(* IEC 61131-3 sources: RL_MAR/experiments/comparison/llm4plc/results/Qwen-Qwen3.5-9B_20260506_150728/20260506_164223, 4 files *)

(* ---- generated_code_iteration_0.st ---- *)
START_ST
FUNCTION_BLOCK RoboticArmColorSorting
VAR_INPUT
    ColorSensorRed : BOOL;   (* Input: Red color sensor *)
    ColorSensorGreen : BOOL;  (* Input: Green color sensor *)
    ColorSensorBlue : BOOL;   (* Input: Blue color sensor *)
END_VAR

VAR_OUTPUT
    RoboticArmMove : BOOL := FALSE;     (* Output: Control for robotic arm movement *)
    BinRed : BOOL := FALSE;           (* Output: Activate red bin *)
    BinGreen : BOOL := FALSE;         (* Output: Activate green bin *)
    BinBlue : BOOL := FALSE;          (* Output: Activate blue bin *)
END_VAR

VAR
    currentState : INT := 0; // 0=IDLE, 1=RED, 2=GREEN, 3=BLUE
END_VAR

BEGIN
    (* STATE 0 (IDLE): No color detected *)
    (* Outputs: RoboticArmMove = FALSE, BinRed = FALSE, BinGreen = FALSE, BinBlue = FALSE *)

    (* STATE 1 (SORTING_RED): Red detected *)
    (* Outputs: RoboticArmMove = TRUE, BinRed = TRUE, BinGreen = FALSE, BinBlue = FALSE *)

    (* STATE 2 (SORTING_GREEN): Green detected *)
    (* Outputs: RoboticArmMove = TRUE, BinRed = FALSE, BinGreen = TRUE, BinBlue = FALSE *)

    (* STATE 3 (SORTING_BLUE): Blue detected *)
    (* Outputs: RoboticArmMove = TRUE, BinRed = FALSE, BinGreen = FALSE, BinBlue = TRUE *)

    (* Transition Logic Implementation *)
    (* Priority Order: Red > Green > Blue as per plan note *)
    (* Logic: If input for current state is FALSE, go to IDLE.
       If input for a different state is TRUE, transition to that new state.
       If input for current state is TRUE, remain in state. *)

    (* Transition from STATE 0 (IDLE) *)
    IF currentState = 0 THEN
        IF ColorSensorRed THEN
            (* Transition 0 -> 1: Red detected *)
            currentState := 1;
        ELSIF ColorSensorGreen THEN
            (* Transition 0 -> 2: Green detected *)
            currentState := 2;
        ELSIF ColorSensorBlue THEN
            (* Transition 0 -> 3: Blue detected *)
            currentState := 3;
        END_IF;
    END_IF;

    (* Transition from STATE 1 (SORTING_RED) *)
    IF currentState = 1 THEN
        IF NOT ColorSensorRed THEN
            (* Transition 1 -> 0: Red sensor lost *)
            currentState := 0;
        ELSIF ColorSensorGreen THEN
            (* Transition 1 -> 2: Green detected while in Red state *)
            currentState := 2;
        ELSIF ColorSensorBlue THEN
            (* Transition 1 -> 3: Blue detected while in Red state *)
            currentState := 3;
        END_IF;
    END_IF;

    (* Transition from STATE 2 (SORTING_GREEN) *)
    IF currentState = 2 THEN
        IF NOT ColorSensorGreen THEN
            (* Transition 2 -> 0: Green sensor lost *)
            currentState := 0;
        ELSIF ColorSensorRed THEN
            (* Transition 2 -> 1: Red detected while in Green state *)
            currentState := 1;
        ELSIF ColorSensorBlue THEN
            (* Transition 2 -> 3: Blue detected while in Green state *)
            currentState := 3;
        END_IF;
    END_IF;

    (* Transition from STATE 3 (SORTING_BLUE) *)
    IF currentState = 3 THEN
        IF NOT ColorSensorBlue THEN
            (* Transition 3 -> 0: Blue sensor lost *)
            currentState := 0;
        ELSIF ColorSensorRed THEN
            (* Transition 3 -> 1: Red detected while in Blue state *)
            currentState := 1;
        ELSIF ColorSensorGreen THEN
            (* Transition 3 -> 2: Green detected while in Blue state *)
            currentState := 2;
        END_IF;
    END_IF;

    (* Assign Outputs based on Final Current State *)
    CASE currentState OF
        0: (* IDLE *)
            RoboticArmMove := FALSE;
            BinRed := FALSE;
            BinGreen := FALSE;
            BinBlue := FALSE;
        1: (* SORTING_RED *)
            RoboticArmMove := TRUE;
            BinRed := TRUE;
            BinGreen := FALSE;
            BinBlue := FALSE;
        2: (* SORTING_GREEN *)
            RoboticArmMove := TRUE;
            BinRed := FALSE;
            BinGreen := TRUE;
            BinBlue := FALSE;
        3: (* SORTING_BLUE *)
            RoboticArmMove := TRUE;
            BinRed := FALSE;
            BinGreen := FALSE;
            BinBlue := TRUE;
    END_CASE;

END_FUNCTION_BLOCK
END_ST

(* ---- generated_code_iteration_2.st ---- *)
START_REASON
The previous code generation failed due to a character encoding issue. The error message "illegal multibyte sequence" at position 78 indicates that the string literal comments (e.g., `(* IDLE *)`) contained non-ASCII characters (likely Chinese characters like "空闲", "分拣", etc., which were not properly escaped or encoded in the UTF-8/ASCII context required by the ANTLR parser and CODESYS compiler).

The compiler expects standard ASCII characters within string literals and comments. To fix this, I will:
1.  Remove all non-ASCII characters from the code, including comments.
2.  Replace descriptive Chinese comments with standard English keywords or simple ASCII placeholders.
3.  Ensure the logic remains identical to the previous iteration (using `CASE` statements for state transitions to avoid the previous "IF" syntax error, and ensuring all semicolons are correctly placed).
4.  Verify that all variable declarations and block structures (`FUNCTION_BLOCK`, `VAR_INPUT`, `VAR_OUTPUT`, `VAR`, `BEGIN`, `END`) are syntactically correct according to IEC 61131-3.

The logic will be:
-   **State 0 (Idle):** If Red -> State 1; If Green -> State 2; If Blue -> State 3.
-   **State 1 (Sort Red):** If Red not detected -> State 0; If Green -> State 2; If Blue -> State 3.
-   **State 2 (Sort Green):** If Green not detected -> State 0; If Red -> State 1; If Blue -> State 3.
-   **State 3 (Sort Blue):** If Blue not detected -> State 0; If Red -> State 1; If Green -> State 2.
-   **Outputs:** Set `RoboticArmMove` and the corresponding `Bin` output based on the final `currentState`.

This approach ensures the code is valid ST, free of encoding errors, and robust against the specific parser issues encountered previously.
END_REASON
START_ST
FUNCTION_BLOCK RoboticArmColorSorting
VAR_INPUT
    ColorSensorRed : BOOL;
    ColorSensorGreen : BOOL;
    ColorSensorBlue : BOOL;
END_VAR

VAR_OUTPUT
    RoboticArmMove : BOOL := FALSE;
    BinRed : BOOL := FALSE;
    BinGreen : BOOL := FALSE;
    BinBlue : BOOL := FALSE;
END_VAR

VAR
    currentState : INT := 0;
END_VAR

BEGIN
    (* Transition Logic *)
    CASE currentState OF
        0:
            IF ColorSensorRed THEN
                currentState := 1;
            ELSIF ColorSensorGreen THEN
                currentState := 2;
            ELSIF ColorSensorBlue THEN
                currentState := 3;
            END_IF;
        1:
            IF NOT ColorSensorRed THEN
                currentState := 0;
            ELSIF ColorSensorGreen THEN
                currentState := 2;
            ELSIF ColorSensorBlue THEN
                currentState := 3;
            END_IF;
        2:
            IF NOT ColorSensorGreen THEN
                currentState := 0;
            ELSIF ColorSensorRed THEN
                currentState := 1;
            ELSIF ColorSensorBlue THEN
                currentState := 3;
            END_IF;
        3:
            IF NOT ColorSensorBlue THEN
                currentState := 0;
            ELSIF ColorSensorRed THEN
                currentState := 1;
            ELSIF ColorSensorGreen THEN
                currentState := 2;
            END_IF;
    END_CASE;

    (* Output Assignment *)
    CASE currentState OF
        0:
            RoboticArmMove := FALSE;
            BinRed := FALSE;
            BinGreen := FALSE;
            BinBlue := FALSE;
        1:
            RoboticArmMove := TRUE;
            BinRed := TRUE;
            BinGreen := FALSE;
            BinBlue := FALSE;
        2:
            RoboticArmMove := TRUE;
            BinRed := FALSE;
            BinGreen := TRUE;
            BinBlue := FALSE;
        3:
            RoboticArmMove := TRUE;
            BinRed := FALSE;
            BinGreen := FALSE;
            BinBlue := TRUE;
    END_CASE;

END_FUNCTION_BLOCK
END_ST

(* ---- generated_code_iteration_3.st ---- *)
START_REASON
The previous code failed the CODESYS compiler validation with the error "应该用';' 替换'CASE'" (Should replace 'CASE' with ';'). This indicates that the compiler does not support the `CASE` statement for state machine transitions in this specific context or version, or it expects a different syntax for state transitions (likely using `IF` statements with explicit state checks or a specific state machine library pattern).

To resolve this, I will replace the `CASE` statements used for state transitions with a series of `IF` statements. The logic will remain:
1.  Check if the current state matches the desired next state based on sensor inputs.
2.  Update `currentState` only if the condition is met.
3.  Keep the second `CASE` statement for output assignment if it is valid, or convert it to `IF` if necessary. However, standard IEC 61131-3 allows `CASE` for discrete variables like `currentState`. The error specifically mentions replacing `CASE` with `;`. This is a very unusual error message for a standard `CASE` statement unless the compiler is misinterpreting the keyword or the project settings are restricted.

Given the strict error message "Replace 'CASE' with ';'", the most robust fix that adheres to the compiler's apparent requirement is to eliminate all `CASE` keywords and replace them with `IF` statements. This ensures maximum compatibility and removes the specific token causing the failure.

Revised Logic:
-   Use `IF currentState = 0 AND ... THEN currentState := 1; END_IF;` pattern for transitions.
-   Use `IF currentState = 1 AND ... THEN currentState := 0; END_IF;` etc.
-   For outputs, use `IF currentState = 1 THEN ... END_IF;` pattern to be safe, though `CASE` is standard for outputs. I will convert the output section to `IF` as well to be absolutely certain no `CASE` keyword triggers the error.

This approach guarantees the code runs without the specific "CASE" keyword error.
END_REASON
START_ST
FUNCTION_BLOCK RoboticArmColorSorting
VAR_INPUT
    ColorSensorRed : BOOL;
    ColorSensorGreen : BOOL;
    ColorSensorBlue : BOOL;
END_VAR

VAR_OUTPUT
    RoboticArmMove : BOOL := FALSE;
    BinRed : BOOL := FALSE;
    BinGreen : BOOL := FALSE;
    BinBlue : BOOL := FALSE;
END_VAR

VAR
    currentState : INT := 0;
END_VAR

BEGIN
    (* Transition Logic - Replaced CASE with IF to fix compiler error *)
    IF currentState = 0 THEN
        IF ColorSensorRed THEN
            currentState := 1;
        ELSIF ColorSensorGreen THEN
            currentState := 2;
        ELSIF ColorSensorBlue THEN
            currentState := 3;
        END_IF;
    END_IF;

    IF currentState = 1 THEN
        IF NOT ColorSensorRed THEN
            currentState := 0;
        ELSIF ColorSensorGreen THEN
            currentState := 2;
        ELSIF ColorSensorBlue THEN
            currentState := 3;
        END_IF;
    END_IF;

    IF currentState = 2 THEN
        IF NOT ColorSensorGreen THEN
            currentState := 0;
        ELSIF ColorSensorRed THEN
            currentState := 1;
        ELSIF ColorSensorBlue THEN
            currentState := 3;
        END_IF;
    END_IF;

    IF currentState = 3 THEN
        IF NOT ColorSensorBlue THEN
            currentState := 0;
        ELSIF ColorSensorRed THEN
            currentState := 1;
        ELSIF ColorSensorGreen THEN
            currentState := 2;
        END_IF;
    END_IF;

    (* Output Assignment - Replaced CASE with IF to fix compiler error *)
    IF currentState = 0 THEN
        RoboticArmMove := FALSE;
        BinRed := FALSE;
        BinGreen := FALSE;
        BinBlue := FALSE;
    END_IF;

    IF currentState = 1 THEN
        RoboticArmMove := TRUE;
        BinRed := TRUE;
        BinGreen := FALSE;
        BinBlue := FALSE;
    END_IF;

    IF currentState = 2 THEN
        RoboticArmMove := TRUE;
        BinRed := FALSE;
        BinGreen := TRUE;
        BinBlue := FALSE;
    END_IF;

    IF currentState = 3 THEN
        RoboticArmMove := TRUE;
        BinRed := FALSE;
        BinGreen := FALSE;
        BinBlue := TRUE;
    END_IF;

END_FUNCTION_BLOCK
END_ST

(* ---- generated_code_iteration_1.st ---- *)
START_REASON
The validation feedback indicates a specific syntax error: "应该用';' 替换'IF'" (Should replace 'IF' with ';'). This is a common issue in IEC 61131-3 Structured Text (ST) when using certain compilers or strict parsers that do not support the `IF` statement as a standalone executable statement without an explicit `THEN` clause in specific contexts, or more likely, the parser expects a semicolon after the condition if it's being treated as a simple expression in a specific dialect, although standard ST requires `IF condition THEN ... END_IF`.

However, looking closely at the error message "replace 'IF' with ';'", it strongly suggests that the compiler is misinterpreting the `IF` keyword or the structure is being parsed incorrectly. In some strict implementations or specific toolchains (like older CODESYS versions or specific embedded compilers), if a block is not properly recognized as a control structure, it might fail.

But the most probable cause for this specific error message in a context where the code looks syntactically correct to a human is that the toolchain expects the `IF` statements to be part of a larger expression or there is a missing semicolon after the condition in a specific dialect, OR (more likely in automated validation tools) the tool is flagging the `IF` keyword itself because it expects a semicolon to terminate a statement if it's not inside a `BEGIN...END` block, but here we are inside `BEGIN`.

Wait, re-reading the error: "replace 'IF' with ';'". This is extremely specific. It often happens when the code is parsed as a sequence of statements where `IF` is expected to be an expression ending in `;`, but `IF` is a keyword. However, in standard ST, `IF condition THEN ... END_IF` is the correct form.

Let's reconsider the error. If the tool says "replace 'IF' with ';'", it might be interpreting the line `IF currentState = 0 THEN` as a statement that needs a semicolon after the condition if it were an expression, but it's a keyword.

Actually, there is a known issue in some strict ST parsers where if you have multiple `IF` statements in sequence, they must be separated by semicolons if they are not part of an `ELSIF` chain, OR the parser is confused by the lack of a semicolon after the `THEN` clause in some dialects (though standard is `THEN`).

Let's look at the structure again.
`IF currentState = 0 THEN`
In standard IEC 61131-3, this is correct.
However, if the error says "replace 'IF' with ';'", it implies the parser thinks `IF` is a variable or an expression that needs a semicolon.

Hypothesis: The specific CODESYS version or the ANTLR grammar used by the validator might require a semicolon after the condition if it's not immediately followed by `THEN` in a specific way, OR it's a false positive due to the `END_IF` placement.

But the most robust fix for "replace 'IF' with ';'" in a context where `IF` is clearly a keyword is to ensure that every statement ends with a semicolon. In ST, `IF ... THEN ... END_IF` is a compound statement. However, if the validator is treating the `IF` line as a standalone statement, it might want a semicolon.

Let's try a different approach. The error might be related to the fact that `IF` is being used without `THEN` in the parser's eyes? No, `THEN` is there.

Let's look at the error again: "应该用';' 替换'IF'". This translates to "Should use ';' to replace 'IF'". This is very strange for standard ST.
Could it be that the tool expects `CASE` statements to be used instead of multiple `IF`s? No, the error specifically mentions `IF`.

Let's consider the possibility that the validator is strict about semicolons after every line, including the `IF` condition line if it's not part of a `CASE` or `WHILE` loop in a specific dialect.
Actually, in some strict implementations, if you have:
`IF cond THEN`
It is correct.
But if the error says replace `IF` with `;`, it might mean the line should be `;`? That makes no sense.

Alternative interpretation: The error message is generated because the parser sees `IF` where it expects an expression ending in `;`. This happens if the `THEN` is missing or if the parser is in a state where it expects an expression.
Wait, if I look at the code:
`IF currentState = 0 THEN`
Maybe the issue is that the validator expects the `IF` statement to be terminated with a semicolon *after* the `THEN`? No, standard is `THEN`.

Let's try to simplify the logic to avoid potential parser ambiguity. We can use `CASE` for the state machine transitions as well, or ensure every line ends with a semicolon if the dialect requires it.
However, the most likely fix for a "replace IF with ;" error in a context like this is that the specific compiler version being used (perhaps an older or non-standard one) does not support the `IF ... THEN` block structure in the way it's written, or it expects the `IF` to be followed by a semicolon if it's a simple statement (which it isn't).

Actually, there is a known quirk in some ST parsers where if you have nested `IF`s or multiple `IF`s, they need to be separated. But here they are sequential.

Let's assume the error is a strict requirement for semicolons after every statement, including the `IF` condition line if the parser treats it as a statement before `THEN`.
So, `IF currentState = 0; THEN`? No, that's invalid ST.
Maybe the error means "The line starting with IF is invalid, replace the IF keyword with a semicolon"? That would mean removing the IF block? No.

Let's reconsider the error message source. "CODESYS: ST output failed...".
In CODESYS, `IF condition THEN` is standard.
Is it possible the user's code has `IF` without `THEN`? No, it has `THEN`.
Is it possible the `THEN` is missing? No.

Wait, could the error be about the `END_IF`? No, it says replace `IF`.

Let's try to rewrite the logic using `CASE` for the transitions to avoid the `IF` keyword entirely, as `CASE` is often preferred for state machines and might bypass this specific parser error if the parser is buggy regarding `IF`.
Or, perhaps the error is a false positive and the real issue is that the `IF` statements are not properly closed or the structure is ambiguous.

Let's try to add semicolons after the conditions if the dialect requires it, or restructure.
Actually, looking at similar issues online, sometimes adding a semicolon after the `IF` condition (before `THEN`) is NOT allowed.
But if the error says "replace IF with ;", it might mean the line `IF currentState = 0 THEN` should be `;`? No.

Let's assume the error is due to the specific toolchain expecting `IF` to be an expression.
Maybe the fix is to use `CASE` for the state transitions?
State 0:
`CASE currentState OF 0: ...`
This avoids `IF`.

Let's try to convert the `IF` blocks to `CASE` blocks for the state transitions. This is a robust way to fix state machine logic in ST and might resolve the `IF` specific error.

Revised Plan:
1. Keep the `VAR` sections.
2. Replace the nested `IF` statements for state transitions with `CASE` statements on `currentState`.
3. Inside the `CASE`, use `IF` for the sensor checks (which are simple conditions) or keep them as `IF` but ensure they are valid.
4. Ensure all `END_CASE` and `END_IF` are present.
5. Ensure the `CASE` statement handles all states (0, 1, 2, 3).

This approach eliminates the problematic `IF currentState = X THEN` pattern which might be triggering the "replace IF with ;" error in the specific validator.

START_ST
FUNCTION_BLOCK RoboticArmColorSorting
VAR_INPUT
    ColorSensorRed : BOOL;
    ColorSensorGreen : BOOL;
    ColorSensorBlue : BOOL;
END_VAR

VAR_OUTPUT
    RoboticArmMove : BOOL := FALSE;
    BinRed : BOOL := FALSE;
    BinGreen : BOOL := FALSE;
    BinBlue : BOOL := FALSE;
END_VAR

VAR
    currentState : INT := 0;
END_VAR

BEGIN
    (* Transition Logic Implementation using CASE for robustness *)
    CASE currentState OF
        0: (* IDLE *)
            IF ColorSensorRed THEN
                currentState := 1;
            ELSIF ColorSensorGreen THEN
                currentState := 2;
            ELSIF ColorSensorBlue THEN
                currentState := 3;
            END_IF;
        1: (* SORTING_RED *)
            IF NOT ColorSensorRed THEN
                currentState := 0;
            ELSIF ColorSensorGreen THEN
                currentState := 2;
            ELSIF ColorSensorBlue THEN
                currentState := 3;
            END_IF;
        2: (* SORTING_GREEN *)
            IF NOT ColorSensorGreen THEN
                currentState := 0;
            ELSIF ColorSensorRed THEN
                currentState := 1;
            ELSIF ColorSensorBlue THEN
                currentState := 3;
            END_IF;
        3: (* SORTING_BLUE *)
            IF NOT ColorSensorBlue THEN
                currentState := 0;
            ELSIF ColorSensorRed THEN
                currentState := 1;
            ELSIF ColorSensorGreen THEN
                currentState := 2;
            END_IF;
    END_CASE;

    (* Assign Outputs based on Final Current State *)
    CASE currentState OF
        0: (* IDLE *)
            RoboticArmMove := FALSE;
            BinRed := FALSE;
            BinGreen := FALSE;
            BinBlue := FALSE;
        1: (* SORTING_RED *)
            RoboticArmMove := TRUE;
            BinRed := TRUE;
            BinGreen := FALSE;
            BinBlue := FALSE;
        2: (* SORTING_GREEN *)
            RoboticArmMove := TRUE;
            BinRed := FALSE;
            BinGreen := TRUE;
            BinBlue := FALSE;
        3: (* SORTING_BLUE *)
            RoboticArmMove := TRUE;
            BinRed := FALSE;
            BinGreen := FALSE;
            BinBlue := TRUE;
    END_CASE;

END_FUNCTION_BLOCK
END_ST
END_REASON
